(* IEC 61131-3 sources: moqui-plc/iec61131/moqui/framework/src/test/pnp, 17 files *)

(* ---- PickAndPlaceFixture.dut ---- *)
(*#-#-#-#-#-#-#-#-#-#---Declaration---#-#-#-#-#-#-#-#-#-#-#-#-#*)

(* Shared fixture for the pick-and-place test suite *)
TYPE PickAndPlaceFixture : STRUCT
    (* Tripod individual-axis enable flags *)
    tripod1Enable : BOOL;
    tripod2Enable : BOOL;
    tripod3Enable : BOOL;

    (* Tripod coordinated group enable flag *)
    tripodEnable : BOOL;

    (* Drive enable flags *)
    rotaryTableEnable : BOOL;
    conveyorEnable : BOOL;

    (* Tripod TCP position - mirrored from AxisGroup.actualPosition each scan. *)
    tripodActualPos : SM3_Robotics.SMC_POS_REF;

    (* Robot FSM flags *)
    robotState : INT;
    readyForMotion : BOOL; (* Group not in Disabled or ErrorStop *)
    ringAttached : BOOL; (* TRUE while robotState ∈ [70..100] *)
    dontChangePCS_2 : BOOL; (* TRUE while robotState ∈ [90..110] *)
    targetConePtr : POINTER TO Cone; (* Cone targeted during ring-place *)

    (* Environment / conveyor state *)
    activeConePtr : POINTER TO Cone; (* Cone currently defining PCS_2 *)
    ringOnTable : BOOL; (* TRUE if any ring is on the table *)

    (*
     * Coordinate-transform gate.
     * Set TRUE by TripodRobot after MC_SetCoordinateTransform.Done.
     * Prevents re-execution after successful setup.
     *)
    coordTransformDone : BOOL;

    (* Process control flags *)
    automaticPnp : BOOL; (* Continuous automatic pick-and-place cycle *)
    setRing : BOOL; (* Manual one-shot ring release *)

    (* Ring FSM diagnostics - written by Environment each scan *)
    ring1State : DINT;
    ring1TrtDone : BOOL;
    ring1TrtError : BOOL;

    (* Rotary table drive diagnostics - written by Environment each scan *)
    rotaryTableAxisReady : BOOL; (* MC_Power.Status *)
    rotaryTableAxisError : BOOL; (* MC_Power.Error *)
END_STRUCT END_TYPE

(* ---- PickAndPlaceFixture.st ---- *)
(* Shared fixture for the pick-and-place test suite *)
TYPE PickAndPlaceFixture : STRUCT
    (* Tripod individual-axis enable flags *)
    tripod1Enable : BOOL;
    tripod2Enable : BOOL;
    tripod3Enable : BOOL;

    (* Tripod coordinated group enable flag *)
    tripodEnable : BOOL;

    (* Drive enable flags *)
    rotaryTableEnable : BOOL;
    conveyorEnable : BOOL;

    (* Tripod TCP position - mirrored from AxisGroup.actualPosition each scan. *)
    tripodActualPos : SM3_Robotics.SMC_POS_REF;

    (* Robot FSM flags *)
    robotState : INT;
    readyForMotion : BOOL; (* Group not in Disabled or ErrorStop *)
    ringAttached : BOOL; (* TRUE while robotState in [70..100] *)
    dontChangePCS_2 : BOOL; (* TRUE while robotState in [90..110] *)
    targetConePtr : POINTER TO Cone; (* Cone targeted during ring-place *)

    (* Environment / conveyor state *)
    activeConePtr : POINTER TO Cone; (* Cone currently defining PCS_2 *)
    ringOnTable : BOOL; (* TRUE if any ring is on the table *)

    (*
     * Coordinate-transform gate.
     * Set TRUE by TripodRobot after MC_SetCoordinateTransform.Done.
     * Prevents re-execution after successful setup.
     *)
    coordTransformDone : BOOL;

    (* Process control flags *)
    automaticPnp : BOOL; (* Continuous automatic pick-and-place cycle *)
    setRing : BOOL; (* Manual one-shot ring release *)

    (* Ring FSM diagnostics - written by Environment each scan *)
    ring1State : DINT;
    ring1TrtDone : BOOL;
    ring1TrtError : BOOL;

    (* Rotary table drive diagnostics - written by Environment each scan *)
    rotaryTableAxisReady : BOOL; (* MC_Power.Status *)
    rotaryTableAxisError : BOOL; (* MC_Power.Error *)
END_STRUCT END_TYPE

(* ---- PickAndPlaceConsts.gvl ---- *)
(*#-#-#-#-#-#-#-#-#-#---Declaration---#-#-#-#-#-#-#-#-#-#-#-#-#*)

VAR_GLOBAL CONSTANT
    (* Tripod MCS origin - machine-frame → tripod-base transform [mm] *)
    tripodTransX : LREAL := 0;
    tripodTransY : LREAL := 0;
    tripodTransZ : LREAL := 1700;
    tripodSize : LREAL := 180;

    (* Conveyor belt MCS offset *)
    beltTransX : LREAL := 0;
    beltTransY : LREAL := 500;
    beltTransZ : LREAL := 0;

    (* Rotary table MCS offset *)
    tableTransX : LREAL := 0;
    tableTransY : LREAL := -500;
    tableTransZ : LREAL := 0;

    (* TCP offset to bottom of ring (ring thickness + gripper) [mm] *)
    tcpRing : LREAL := 0.02 * tripodSize + 15; (* ≈ 18.6 mm *)

    (* Tripod initial slider positions [mm] *)
    tripod1PosOrig : REAL := 50;
    tripod2PosOrig : REAL := 75;
    tripod3PosOrig : REAL := 25;

    (* Tripod group dynamics *)
    tripodVelocity : LREAL := 1000; (* [mm/s] *)
    tripodAcceleration : LREAL :=  10000; (* [mm/s²] *)
    tripodJerk : LREAL := 100000; (* [mm/s³] *)

    (* Rotary-table drive dynamics *)
    tableVelocity : LREAL :=  50; (* [°/s] *)
    tableAcceleration : LREAL :=  30; (* [°/s²] *)

    (* Conveyor belt drive dynamics *)
    beltVelocity : LREAL := 300; (* [mm/s] *)
    beltAcceleration : LREAL := 150; (* [mm/s²] *)
END_VAR

(* ---- PickAndPlaceConsts.st ---- *)
VAR_GLOBAL CONSTANT
    (* Tripod MCS origin - machine-frame -> tripod-base transform [mm] *)
    tripodTransX : LREAL := 0;
    tripodTransY : LREAL := 0;
    tripodTransZ : LREAL := 1700;
    tripodSize : LREAL := 180;

    (* Conveyor belt MCS offset *)
    beltTransX : LREAL := 0;
    beltTransY : LREAL := 500;
    beltTransZ : LREAL := 0;

    (* Rotary table MCS offset *)
    tableTransX : LREAL := 0;
    tableTransY : LREAL := -500;
    tableTransZ : LREAL := 0;

    (* TCP offset to bottom of ring (ring thickness + gripper) [mm] *)
    tcpRing : LREAL := 0.02 * tripodSize + 15; (* ~= 18.6 mm *)

    (* Tripod initial slider positions [mm] *)
    tripod1PosOrig : REAL := 50;
    tripod2PosOrig : REAL := 75;
    tripod3PosOrig : REAL := 25;

    (* Tripod group dynamics *)
    tripodVelocity : LREAL := 1000; (* [mm/s] *)
    tripodAcceleration : LREAL :=  10000; (* [mm/s²] *)
    tripodJerk : LREAL := 100000; (* [mm/s³] *)

    (* Rotary-table drive dynamics *)
    tableVelocity : LREAL :=  50; (* [°/s] *)
    tableAcceleration : LREAL :=  30; (* [°/s²] *)

    (* Conveyor belt drive dynamics *)
    beltVelocity : LREAL := 300; (* [mm/s] *)
    beltAcceleration : LREAL := 150; (* [mm/s²] *)
END_VAR

(* ---- PickAndPlaceData.gvl ---- *)
(*#-#-#-#-#-#-#-#-#-#---Declaration---#-#-#-#-#-#-#-#-#-#-#-#-#*)

VAR_GLOBAL
    (* Test suite fixture *)
    pnp : PickAndPlaceFixture;
END_VAR

(* ---- PickAndPlaceData.st ---- *)
VAR_GLOBAL
    (* Test suite fixture *)
    pnp : PickAndPlaceFixture;
END_VAR

(* ---- Cone.pou ---- *)
(*#-#-#-#-#-#-#-#-#-#---Declaration---#-#-#-#-#-#-#-#-#-#-#-#-#*)

(* Conveyor-belt cone tracking.
 *
 * FSM:
 *   0   Invisible - waits until previous cone is on belt and far enough,
 *       or 'start' input fires (bootstrap for the first cone)
 *   10  Linking PCS_2 to cone position via MC_TrackConveyorBelt
 *   20  Cone on belt - tracks position until exit point reached
 *)
FUNCTION_BLOCK Cone
VAR_EXTERNAL
	pnp : PickAndPlaceFixture;
END_VAR
VAR_IN_OUT
	activeConePtr : POINTER TO Cone; (* Written to this when cone becomes active *)
END_VAR
VAR_INPUT
	previousConePtr : POINTER TO Cone; (* Previous cone in the circular chain *)
	start : BOOL;
END_VAR
VAR_OUTPUT
	pos : SM3_Robotics.MC_COORD_REF;
	state : DINT;
	onBelt : BOOL;
END_VAR
VAR
	conveyorBeltOrigin : SM3_Robotics.MC_COORD_REF :=
		(X := beltTransX, Y := beltTransY, Z := beltTransZ);
	initialConePosition : SM3_Robotics.MC_COORD_REF := (X := -925, Z := 125);
	tcb : SM3_Robotics.MC_TrackConveyorBelt := (
		ConveyorBeltOrigin := conveyorBeltOrigin,
		InitialObjectPosition := initialConePosition,
		CoordSystem := SM3_Robotics.SMC_COORD_SYSTEM.PCS_2);
	frame : SM3_Robotics.SMC_Frame;
	stateOld : DINT;
END_VAR

(*#-#-#-#-#-#-#-#-#-#---Implementation---#-#-#-#-#-#-#-#-#-#-#-#-#*)

REPEAT
	stateOld := state;

	CASE state OF
		0 :	(* Invisible - wait until the previous cone has advanced sufficiently *)
			IF start OR (NOT pnp.dontChangePCS_2
					AND previousConePtr^.onBelt
					AND previousConePtr^.pos.X >= -250) THEN
				tcb(Execute := FALSE,
					AxisGroup := Tripod,
					ConveyorBelt := DriveConveyorBelt);
				tcb.Execute := TRUE;
				state := state + 10;
			END_IF;

		10 : (* Linking PCS_2 to the position of this cone *)
			IF tcb.Done THEN
				onBelt := TRUE;
				activeConePtr := THIS;
				state := state + 10;
			END_IF;

		20 : (* Cone on belt - track position until it reaches the exit *)
			tcb.cs.GetPose(cs := frame, fTime := Tripod1.fTaskCycle);
			SM3_Robotics.SMC_Frame_To_CoordRef(c := pos, f := frame);
			IF pos.X >= beltTransX + 725 THEN
				onBelt := FALSE;
				state := 0;
			END_IF;
	END_CASE;

	tcb(AxisGroup := Tripod, ConveyorBelt := DriveConveyorBelt);
UNTIL state = stateOld END_REPEAT

(* ---- Cone.st ---- *)
(* Conveyor-belt cone tracking.
 *
 * FSM:
 *   0   Invisible - waits until previous cone is on belt and far enough,
 *       or 'start' input fires (bootstrap for the first cone)
 *   10  Linking PCS_2 to cone position via MC_TrackConveyorBelt
 *   20  Cone on belt - tracks position until exit point reached
 *)
FUNCTION_BLOCK Cone
	VAR_EXTERNAL
		pnp : PickAndPlaceFixture;
	END_VAR
	VAR_IN_OUT
		activeConePtr : POINTER TO Cone; (* Written to this when cone becomes active *)
	END_VAR
	VAR_INPUT
		previousConePtr : POINTER TO Cone; (* Previous cone in the circular chain *)
		start : BOOL;
	END_VAR
	VAR_OUTPUT
		pos : SM3_Robotics.MC_COORD_REF;
		state : DINT;
		onBelt : BOOL;
	END_VAR
	VAR
		conveyorBeltOrigin : SM3_Robotics.MC_COORD_REF :=
			(X := beltTransX, Y := beltTransY, Z := beltTransZ);
		initialConePosition : SM3_Robotics.MC_COORD_REF := (X := -925, Z := 125);
		tcb : SM3_Robotics.MC_TrackConveyorBelt := (
			ConveyorBeltOrigin := conveyorBeltOrigin,
			InitialObjectPosition := initialConePosition,
			CoordSystem := SM3_Robotics.SMC_COORD_SYSTEM.PCS_2);
		frame : SM3_Robotics.SMC_Frame;
		stateOld : DINT;
	END_VAR

	REPEAT
		stateOld := state;

		CASE state OF
			0 :	(* Invisible - wait until the previous cone has advanced sufficiently *)
				IF start OR (NOT pnp.dontChangePCS_2
						AND previousConePtr^.onBelt
						AND previousConePtr^.pos.X >= -250) THEN
					tcb(Execute := FALSE,
						AxisGroup := Tripod,
						ConveyorBelt := DriveConveyorBelt);
					tcb.Execute := TRUE;
					state := state + 10;
				END_IF;

			10 : (* Linking PCS_2 to the position of this cone *)
				IF tcb.Done THEN
					onBelt := TRUE;
					activeConePtr := THIS;
					state := state + 10;
				END_IF;

			20 : (* Cone on belt - track position until it reaches the exit *)
				tcb.cs.GetPose(cs := frame, fTime := Tripod1.fTaskCycle);
				SM3_Robotics.SMC_Frame_To_CoordRef(c := pos, f := frame);
				IF pos.X >= beltTransX + 725 THEN
					onBelt := FALSE;
					state := 0;
				END_IF;
		END_CASE;

		tcb(AxisGroup := Tripod, ConveyorBelt := DriveConveyorBelt);
	UNTIL state = stateOld END_REPEAT
	END_FUNCTION_BLOCK

(* ---- Environment.pou ---- *)
(*#-#-#-#-#-#-#-#-#-#---Declaration---#-#-#-#-#-#-#-#-#-#-#-#-#*)

{attribute 'no_assign'}
(* Hardware-abstraction layer for the conveyance environment.
 *
 * Responsibilities:
 *   1. Drive the rotary-table and conveyor-belt axes with MC_Power + MC_MoveVelocity.
 *      (continuous rotation/feed - no homing required for these drives).
 *   2. Run the cone state machines (three cones on the conveyor belt).
 *   3. Run the ring state machines (two rings on the rotary table).
 *   4. Publish activeCone and ringOnTable each scan.
 *)
FUNCTION_BLOCK Environment
VAR_EXTERNAL
	pnp : PickAndPlaceFixture;
END_VAR
VAR_INPUT
	operationType : OperatingMode;
END_VAR
VAR
	(* Drive axes - MC_Power + MC_MoveVelocity, no homing for continuous drives *)
	powRotaryTable : MC_Power := (Enable := TRUE, bRegulatorOn := TRUE, bDriveStart := TRUE);
	powConveyorBelt : MC_Power := (Enable := TRUE, bRegulatorOn := TRUE, bDriveStart := TRUE);
	mvRotaryTable : MC_MoveVelocity := (Execute := TRUE, Velocity := tableVelocity, Acceleration := tableAcceleration, Deceleration := tableAcceleration, Jerk := 1000);
	mvConveyorBelt : MC_MoveVelocity := (Execute := TRUE, Velocity := beltVelocity, Acceleration := beltAcceleration, Deceleration := beltAcceleration, Jerk := 1000);

	(* Cones - three instances on the belt (circular chain) *)
	cone1 : Cone;
	cone2 : Cone;
	cone3 : Cone;

	(* Rings - two instances on the rotary table *)
	ring1 : Ring;
	ring2 : Ring;

	ring1StartPos : SM3_Robotics.MC_COORD_REF := (X :=  75, Y := 100, Z := 0);
	ring2StartPos : SM3_Robotics.MC_COORD_REF := (X := -75, Y := 100, Z := 0);

	init : BOOL := TRUE; (* First-scan bootstrap flag *)
END_VAR

(*#-#-#-#-#-#-#-#-#-#---Implementation---#-#-#-#-#-#-#-#-#-#-#-#-#*)

(* Rotary table and conveyor belt drives - power and continuous velocity *)
powRotaryTable(Axis := DriveRotaryTable);
powConveyorBelt(Axis := DriveConveyorBelt);

(* Drive status diagnostics - updated before the guard so they are visible even if RETURN fires *)
pnp.rotaryTableAxisReady := powRotaryTable.Status;
pnp.rotaryTableAxisError := powRotaryTable.Error;

(* Wait for both drives powered before running cones / rings *)
IF NOT (powRotaryTable.Status AND powConveyorBelt.Status) THEN
	init := TRUE;
	RETURN;
END_IF;
mvRotaryTable(Axis := DriveRotaryTable);
mvConveyorBelt(Axis := DriveConveyorBelt);

(* Wait for the tripod group to be ready before starting cone/ring FSMs *)
IF NOT pnp.readyForMotion THEN
	RETURN;
END_IF;

(* Cone state machines *)
(*
 * cone1.start := init bootstraps the circular chain on the first scan:
 *   cone1 activates immediately (skips the chain-guard condition).
 *   cone2 and cone3 activate in sequence once cone1 advances on the belt.
 *)
cone1(activeConePtr := pnp.activeConePtr, previousConePtr := ADR(cone3), start := init);
cone2(activeConePtr := pnp.activeConePtr, previousConePtr := ADR(cone1), start := FALSE);
cone3(activeConePtr := pnp.activeConePtr, previousConePtr := ADR(cone2), start := FALSE);

(* Ring state machines *)
IF init THEN
	ring1.startPos := ring1StartPos;
	ring2.startPos := ring2StartPos;
END_IF;

ring1(otherRingPtr := ADR(ring2));
ring2(otherRingPtr := ADR(ring1));

(* Publish environment state to pnp *)
pnp.ringOnTable := ring1.onTable OR ring2.onTable;

(* Ring FSM diagnostics *)
pnp.ring1State := ring1.state;
pnp.ring1TrtDone := ring1.trt.Done;
pnp.ring1TrtError := ring1.trt.Error;

init := FALSE;

(* ---- Environment.st ---- *)
(* Hardware-abstraction layer for the conveyance environment.
 *
 * Responsibilities:
 *   1. Drive the rotary-table and conveyor-belt axes with MC_Power + MC_MoveVelocity.
 *      (continuous rotation/feed - no homing required for these drives).
 *   2. Run the cone state machines (three cones on the conveyor belt).
 *   3. Run the ring state machines (two rings on the rotary table).
 *   4. Publish activeCone and ringOnTable each scan.
 *)
FUNCTION_BLOCK Environment
	VAR_EXTERNAL
		pnp : PickAndPlaceFixture;
	END_VAR
	VAR_INPUT
		operationType : OperatingMode;
	END_VAR
	VAR
		(* Drive axes - MC_Power + MC_MoveVelocity, no homing for continuous drives *)
		powRotaryTable : MC_Power := (Enable := TRUE, bRegulatorOn := TRUE, bDriveStart := TRUE);
		powConveyorBelt : MC_Power := (Enable := TRUE, bRegulatorOn := TRUE, bDriveStart := TRUE);
		mvRotaryTable : MC_MoveVelocity := (Execute := TRUE, Velocity := tableVelocity, Acceleration := tableAcceleration, Deceleration := tableAcceleration, Jerk := 1000);
		mvConveyorBelt : MC_MoveVelocity := (Execute := TRUE, Velocity := beltVelocity, Acceleration := beltAcceleration, Deceleration := beltAcceleration, Jerk := 1000);

		(* Cones - three instances on the belt (circular chain) *)
		cone1 : Cone;
		cone2 : Cone;
		cone3 : Cone;

		(* Rings - two instances on the rotary table *)
		ring1 : Ring;
		ring2 : Ring;

		ring1StartPos : SM3_Robotics.MC_COORD_REF := (X :=  75, Y := 100, Z := 0);
		ring2StartPos : SM3_Robotics.MC_COORD_REF := (X := -75, Y := 100, Z := 0);

		init : BOOL := TRUE; (* First-scan bootstrap flag *)
	END_VAR

	(* Rotary table and conveyor belt drives - power and continuous velocity *)
	powRotaryTable(Axis := DriveRotaryTable);
	powConveyorBelt(Axis := DriveConveyorBelt);

	(* Drive status diagnostics - updated before the guard so they are visible even if RETURN fires *)
	pnp.rotaryTableAxisReady := powRotaryTable.Status;
	pnp.rotaryTableAxisError := powRotaryTable.Error;

	(* Wait for both drives powered before running cones / rings *)
	IF NOT (powRotaryTable.Status AND powConveyorBelt.Status) THEN
		init := TRUE;
		RETURN;
	END_IF;
	mvRotaryTable(Axis := DriveRotaryTable);
	mvConveyorBelt(Axis := DriveConveyorBelt);

	(* Wait for the tripod group to be ready before starting cone/ring FSMs *)
	IF NOT pnp.readyForMotion THEN
		RETURN;
	END_IF;

	(* Cone state machines *)
	(*
	 * cone1.start := init bootstraps the circular chain on the first scan:
	 *   cone1 activates immediately (skips the chain-guard condition).
	 *   cone2 and cone3 activate in sequence once cone1 advances on the belt.
	 *)
	cone1(activeConePtr := pnp.activeConePtr, previousConePtr := ADR(cone3), start := init);
	cone2(activeConePtr := pnp.activeConePtr, previousConePtr := ADR(cone1), start := FALSE);
	cone3(activeConePtr := pnp.activeConePtr, previousConePtr := ADR(cone2), start := FALSE);

	(* Ring state machines *)
	IF init THEN
		ring1.startPos := ring1StartPos;
		ring2.startPos := ring2StartPos;
	END_IF;

	ring1(otherRingPtr := ADR(ring2));
	ring2(otherRingPtr := ADR(ring1));

	(* Publish environment state to pnp *)
	pnp.ringOnTable := ring1.onTable OR ring2.onTable;

	(* Ring FSM diagnostics *)
	pnp.ring1State := ring1.state;
	pnp.ring1TrtDone := ring1.trt.Done;
	pnp.ring1TrtError := ring1.trt.Error;

	init := FALSE;
	END_FUNCTION_BLOCK

(* ---- Ring.pou ---- *)
(*#-#-#-#-#-#-#-#-#-#---Declaration---#-#-#-#-#-#-#-#-#-#-#-#-#*)

(* Rotary-table ring tracking.
 *
 * State machine:
 *   0   Ring at start position - waits for safe conditions + trigger
 *   10  Linking PCS_1 to ring via MC_TrackRotaryTable
 *   20  Ring on table, spinning - waits until robot is free
 *   30  Waiting for robot to pick up ring
 *   40  Ring attached to robot - follows TCP position
 *   50  Ring placed on cone - follows cone position until cone leaves belt
 *)
FUNCTION_BLOCK Ring
VAR_EXTERNAL
	pnp : PickAndPlaceFixture;
END_VAR
VAR_INPUT
	otherRingPtr : POINTER TO Ring; (* The other ring in the pair *)
	startPos : SM3_Robotics.MC_COORD_REF; (* Initial position in MCS *)
END_VAR
VAR_OUTPUT
	pos : SM3_Robotics.MC_COORD_REF;
	state  : DINT;
	onTable : BOOL;
END_VAR
VAR
	stateOld : DINT;
	frame : SM3_Robotics.SMC_Frame;
	rotaryTableOrigin : SM3_Robotics.MC_COORD_REF :=
		(X := tableTransX, Y := tableTransY, Z := tableTransZ);
	initialObjectPosition : SM3_Robotics.MC_COORD_REF := (Y := 400, Z := 30);
	trt : SM3_Robotics.MC_TrackRotaryTable := (
		RotaryTableOrigin := rotaryTableOrigin,
		initialObjectPosition := initialObjectPosition,
		CoordSystem := SM3_Robotics.SMC_COORD_SYSTEM.PCS_1);
	conePtr : POINTER TO Cone;
END_VAR

(*#-#-#-#-#-#-#-#-#-#---Implementation---#-#-#-#-#-#-#-#-#-#-#-#-#*)

REPEAT
	stateOld := state;
	CASE state OF

	0 :	(* Ring at start position - wait for safe conditions and cycle trigger *)
		pos := startPos;

		IF pnp.readyForMotion AND (otherRingPtr^.state = 0 OR otherRingPtr^.state >= 40)
				AND (pnp.setRing OR pnp.automaticPnp) THEN
			trt(Execute := FALSE,
			    AxisGroup := Tripod,
			    RotaryTable := DriveRotaryTable);
			trt.Execute := TRUE;
			state := state + 10;
		END_IF;

	10 : (* Linking PCS_1 to the position of this ring *)
		IF trt.Done THEN
			state := state + 10;
		END_IF;

	20 : (* Ring on rotary table, spinning - wait until robot is free to pick *)
		trt.cs.GetPose(cs := frame, fTime := Tripod1.fTaskCycle);
		SM3_Robotics.SMC_Frame_To_CoordRef(c := pos, f := frame);

		IF NOT pnp.ringAttached THEN
			state := state + 10;
		END_IF;

	30 : (* Waiting for robot to attach to ring *)
		trt.cs.GetPose(cs := frame, fTime := Tripod1.fTaskCycle);
		SM3_Robotics.SMC_Frame_To_CoordRef(c := pos, f := frame);

		IF pnp.ringAttached THEN
			state := state + 10;
		END_IF;

	40 : (* Ring attached to robot - follow TCP position *)
		pos.X := pnp.tripodActualPos.c.X;
		pos.Y := pnp.tripodActualPos.c.Y;
		pos.Z := pnp.tripodActualPos.c.Z - tcpRing;

		IF NOT pnp.ringAttached THEN
			conePtr := pnp.targetConePtr;
			state := state + 10;
		END_IF;

	50 : (* Ring placed on cone - follow cone position until cone exits belt *)
		pos.X := conePtr^.pos.X;
		pos.Y := conePtr^.pos.Y;
		pos.Z := conePtr^.pos.Z;

		IF NOT conePtr^.onBelt THEN
			state := 0;
		END_IF;
	END_CASE;

	trt(AxisGroup := Tripod, RotaryTable := DriveRotaryTable);
UNTIL state = stateOld END_REPEAT;

onTable := state = 20 OR state = 30;

(* ---- Ring.st ---- *)
(* Rotary-table ring tracking.
 *
 * State machine:
 *   0   Ring at start position - waits for safe conditions + trigger
 *   10  Linking PCS_1 to ring via MC_TrackRotaryTable
 *   20  Ring on table, spinning - waits until robot is free
 *   30  Waiting for robot to pick up ring
 *   40  Ring attached to robot - follows TCP position
 *   50  Ring placed on cone - follows cone position until cone leaves belt
 *)
FUNCTION_BLOCK Ring
	VAR_EXTERNAL
		pnp : PickAndPlaceFixture;
	END_VAR
	VAR_INPUT
		otherRingPtr : POINTER TO Ring; (* The other ring in the pair *)
		startPos : SM3_Robotics.MC_COORD_REF; (* Initial position in MCS *)
	END_VAR
	VAR_OUTPUT
		pos : SM3_Robotics.MC_COORD_REF;
		state  : DINT;
		onTable : BOOL;
	END_VAR
	VAR
		stateOld : DINT;
		frame : SM3_Robotics.SMC_Frame;
		rotaryTableOrigin : SM3_Robotics.MC_COORD_REF :=
			(X := tableTransX, Y := tableTransY, Z := tableTransZ);
		initialObjectPosition : SM3_Robotics.MC_COORD_REF := (Y := 400, Z := 30);
		trt : SM3_Robotics.MC_TrackRotaryTable := (
			RotaryTableOrigin := rotaryTableOrigin,
			initialObjectPosition := initialObjectPosition,
			CoordSystem := SM3_Robotics.SMC_COORD_SYSTEM.PCS_1);
		conePtr : POINTER TO Cone;
	END_VAR

	REPEAT
		stateOld := state;
		CASE state OF

		0 :	(* Ring at start position - wait for safe conditions and cycle trigger *)
			pos := startPos;

			IF pnp.readyForMotion AND (otherRingPtr^.state = 0 OR otherRingPtr^.state >= 40)
					AND (pnp.setRing OR pnp.automaticPnp) THEN
				trt(Execute := FALSE,
				    AxisGroup := Tripod,
				    RotaryTable := DriveRotaryTable);
				trt.Execute := TRUE;
				state := state + 10;
			END_IF;

		10 : (* Linking PCS_1 to the position of this ring *)
			IF trt.Done THEN
				state := state + 10;
			END_IF;

		20 : (* Ring on rotary table, spinning - wait until robot is free to pick *)
			trt.cs.GetPose(cs := frame, fTime := Tripod1.fTaskCycle);
			SM3_Robotics.SMC_Frame_To_CoordRef(c := pos, f := frame);

			IF NOT pnp.ringAttached THEN
				state := state + 10;
			END_IF;

		30 : (* Waiting for robot to attach to ring *)
			trt.cs.GetPose(cs := frame, fTime := Tripod1.fTaskCycle);
			SM3_Robotics.SMC_Frame_To_CoordRef(c := pos, f := frame);

			IF pnp.ringAttached THEN
				state := state + 10;
			END_IF;

		40 : (* Ring attached to robot - follow TCP position *)
			pos.X := pnp.tripodActualPos.c.X;
			pos.Y := pnp.tripodActualPos.c.Y;
			pos.Z := pnp.tripodActualPos.c.Z - tcpRing;

			IF NOT pnp.ringAttached THEN
				conePtr := pnp.targetConePtr;
				state := state + 10;
			END_IF;

		50 : (* Ring placed on cone - follow cone position until cone exits belt *)
			pos.X := conePtr^.pos.X;
			pos.Y := conePtr^.pos.Y;
			pos.Z := conePtr^.pos.Z;

			IF NOT conePtr^.onBelt THEN
				state := 0;
			END_IF;
		END_CASE;

		trt(AxisGroup := Tripod, RotaryTable := DriveRotaryTable);
	UNTIL state = stateOld END_REPEAT;

	onTable := state = 20 OR state = 30;
	END_FUNCTION_BLOCK

(* ---- TripodRobot.pou ---- *)
(*#-#-#-#-#-#-#-#-#-#---Declaration---#-#-#-#-#-#-#-#-#-#-#-#-#*)

{attribute 'no_assign'}
(* Tripod robot motion FSM using Moqui AxisGroup and Axis wrappers.
 *
 * FSM:
 *   0    Wait for all three tripod axes powered and ready
 *   10   Set initial slider positions (AxisCmd.SetPosition x 3)
 *   20   Set MCS coordinate transform (MC_SetCoordinateTransform, direct)
 *   30   Enable axis group (AxisGroup.groupEnable -> Standby)
 *   40   Wait for ring on table; issue MoveLinearAbsolute to ring (PCS_1)
 *   50   Wait commandExecuted (arrival at ring)
 *   60   Wait 200 ms (ring following), then issue MoveLinearRelative upward (PCS_1)
 *   70   Wait commandExecuted; issue MoveLinearAbsolute to rest (WCS)
 *   80   Wait commandExecuted; [release] then MoveLinearAbsolute above cone (PCS_2)
 *   90   Wait commandExecuted; [release] then MoveLinearAbsolute on cone (PCS_2)
 *   100  Wait commandExecuted; [release] then MoveLinearAbsolute above cone (PCS_2)
 *   110  Wait commandExecuted; [release] then MoveLinearAbsolute to rest (WCS)
 *   120  Wait commandExecuted; [release] then loop to state 40
 *
 * [release] means: the previous command was also MoveLinearAbsolute, so the
 * AxisGroup FSM stays in CheckLinearAbsoluteState (commandExecuted=TRUE) until the caller changes cmd.
 * On commandExecuted, set cmd=Idle -> AxisGroup returns to Standby (ready=TRUE) -> set the new MoveLinearAbsolute target.
 * This 2-scan handshake is needed only when two consecutive commands share the
 * same AxisGroupCmd value (both MoveLinearAbsolute).
 *
 * Unconditional FB calls at the bottom execute every scan regardless of state,
 * following the standard CODESYS PLCopen pattern.
 *)
FUNCTION_BLOCK TripodRobot
VAR_EXTERNAL
	pnp : PickAndPlaceFixture;
END_VAR
VAR_INPUT
	operationType : OperatingMode;
END_VAR
VAR_OUTPUT
	groupError : BOOL;
	groupErrorId : DWORD;
END_VAR
VAR
	(* Tripod individual axes *)
	tripodAxis1 : Axis;
	tripodAxis2 : Axis;
	tripodAxis3 : Axis;

	(* Tripod coordinated group - AxisGroup wraps all Cartesian moves *)
	tripodGroup : AxisGroup;

	(* Coordinate transform - direct PLCopen call *)
	setCoord : SM3_Robotics.MC_SetCoordinateTransform;
	mcs : SM3_Robotics.MC_COORD_REF;

	(* 200ms ring-following timer (state 60) *)
	ton : TON := (PT := T#200MS);

	(*
     * Constant Cartesian target positions.
	 * All X,Y components default to 0 (struct zero-init).
	 * Only Z (and coordinate system) distinguishes them.
     *)
	posAboveRingPCS1 : SM3_Robotics.SMC_POS_REF; (* Z = tcpRing, PCS_1 *)
	posAboveConePCS2 : SM3_Robotics.SMC_POS_REF; (* Z = 200, PCS_2 *)
	posOnConePCS2 : SM3_Robotics.SMC_POS_REF; (* Z = tcpRing, PCS_2 *)
	posRestWCS : SM3_Robotics.SMC_POS_REF; (* Z = 300, WCS *)
END_VAR

(*#-#-#-#-#-#-#-#-#-#---Implementation---#-#-#-#-#-#-#-#-#-#-#-#-#*)

(* Target positions - set each scan (struct re-init on first scan) *)
posAboveRingPCS1.c.Z := tcpRing;
posAboveConePCS2.c.Z := 200;
posOnConePCS2.c.Z := tcpRing;
posRestWCS.c.Z := 300;

(* Tripod robot FSM *)
CASE pnp.robotState OF
	0 : (* Wait for all three tripod axes powered and homed *)
		pnp.tripod1Enable := TRUE;
		pnp.tripod2Enable := TRUE;
		pnp.tripod3Enable := TRUE;
		IF tripodAxis1.ready AND tripodAxis2.ready AND tripodAxis3.ready THEN
			pnp.robotState := 10;
		END_IF

	10 : (* Set initial slider positions *)
		tripodAxis1.cmd := AxisCmd.SetPosition;
		tripodAxis1.position := tripod1PosOrig;
		tripodAxis2.cmd := AxisCmd.SetPosition;
		tripodAxis2.position := tripod2PosOrig;
		tripodAxis3.cmd := AxisCmd.SetPosition;
		tripodAxis3.position := tripod3PosOrig;

		IF tripodAxis1.commandExecuted AND tripodAxis2.commandExecuted
				AND tripodAxis3.commandExecuted THEN
			tripodAxis1.cmd := AxisCmd.Idle;
			tripodAxis2.cmd := AxisCmd.Idle;
			tripodAxis3.cmd := AxisCmd.Idle;
			setCoord.Execute := FALSE; (* Arm rising edge for state 20 *)
			pnp.robotState := 20;
		END_IF;

	20 : (* Set MCS coordinate transform (direct MC_SetCoordinateTransform) *)
		mcs.X := tripodTransX;
		mcs.Y := tripodTransY;
		mcs.Z := tripodTransZ;
		setCoord.Execute := TRUE;
		setCoord.CoordTransform := mcs;
		setCoord.CoordSystem := SM3_Robotics.SMC_COORD_SYSTEM.MCS;

		IF setCoord.Done THEN
			pnp.coordTransformDone := TRUE;
			pnp.robotState := 30;
		END_IF;

	30 : (* Enable axis group - AxisGroup transitions to Standby *)
		pnp.tripodEnable := TRUE;

		IF tripodGroup.ready THEN
			pnp.robotState := 40;
		END_IF;

	40 : (* Wait for ring on table, then issue move to ring (PCS_1) *)
		IF pnp.ringOnTable THEN
			tripodGroup.cmd := AxisGroupCmd.MoveLinearAbsolute;
			tripodGroup.endPoint := posAboveRingPCS1;
			tripodGroup.coordinateSystem := SM3_Robotics.SMC_COORD_SYSTEM.PCS_1;
			tripodGroup.velocity := tripodVelocity;
			tripodGroup.acceleration := tripodAcceleration;
			tripodGroup.deceleration := tripodAcceleration;
			tripodGroup.jerk := tripodJerk;
			tripodGroup.bufferMode := SM3_Basic.MC_BUFFER_MODE.BlendingHigh;
			tripodGroup.transitionMode := SM3_Robotics.MC_TRANSITION_MODE.TMCornerDistance;
			tripodGroup.transitionParameter := 500;
			pnp.robotState := 50;
		END_IF;

	50 : (* Wait for arrival at ring *)
		IF tripodGroup.commandExecuted THEN
			ton(IN := FALSE); (* Reset 200 ms timer *)
			pnp.robotState := 60;
		END_IF;

	60 : (* Wait 200 ms following the ring, then move upward *)
		ton(IN := TRUE);

		IF ton.Q THEN
			tripodGroup.cmd := AxisGroupCmd.MoveLinearRelative;
			tripodGroup.endPoint.c.X := 0;
			tripodGroup.endPoint.c.Y := 0;
			tripodGroup.endPoint.c.Z := 150;
			tripodGroup.coordinateSystem := SM3_Robotics.SMC_COORD_SYSTEM.WCS;
			tripodGroup.bufferMode := SM3_Basic.MC_BUFFER_MODE.Buffered;
			tripodGroup.transitionMode := SM3_Robotics.MC_TRANSITION_MODE.TMNone;
			tripodGroup.transitionParameter := 0;
			pnp.robotState := 70;
		END_IF;

	70 : (* Queue MoveLinearAbsolute to rest (WCS), matching the sample's buffered handoff *)
		tripodGroup.cmd := AxisGroupCmd.MoveLinearAbsolute;
		tripodGroup.endPoint := posRestWCS;
		tripodGroup.coordinateSystem := SM3_Robotics.SMC_COORD_SYSTEM.WCS;
		tripodGroup.bufferMode := SM3_Basic.MC_BUFFER_MODE.BlendingHigh;
		tripodGroup.transitionMode := SM3_Robotics.MC_TRANSITION_MODE.TMCornerDistance;
		tripodGroup.transitionParameter := 500;
		pnp.robotState := 80;

	80 : (* [release] wait rest-pos done; then move above cone (PCS_2) *)
		IF tripodGroup.commandExecuted THEN
			tripodGroup.cmd := AxisGroupCmd.Idle;
		ELSIF tripodGroup.ready THEN
			pnp.targetConePtr := pnp.activeConePtr;
			tripodGroup.cmd := AxisGroupCmd.MoveLinearAbsolute;
			tripodGroup.endPoint := posAboveConePCS2;
			tripodGroup.coordinateSystem := SM3_Robotics.SMC_COORD_SYSTEM.PCS_2;
			tripodGroup.bufferMode := SM3_Basic.MC_BUFFER_MODE.aborting;
			tripodGroup.transitionMode := SM3_Robotics.MC_TRANSITION_MODE.TMNone;
			tripodGroup.transitionParameter := 0;
			pnp.robotState := 90;
		END_IF;

	90 : (* [release] wait above-cone done; then move down to cone (PCS_2) *)
		IF tripodGroup.commandExecuted THEN
			tripodGroup.cmd := AxisGroupCmd.Idle;
		ELSIF tripodGroup.ready THEN
			tripodGroup.cmd := AxisGroupCmd.MoveLinearAbsolute;
			tripodGroup.endPoint := posOnConePCS2;
			tripodGroup.coordinateSystem := SM3_Robotics.SMC_COORD_SYSTEM.PCS_2;
			tripodGroup.bufferMode := SM3_Basic.MC_BUFFER_MODE.aborting;
			tripodGroup.transitionMode := SM3_Robotics.MC_TRANSITION_MODE.TMNone;
			tripodGroup.transitionParameter := 0;
			pnp.robotState := 100;
		END_IF;

	100 : (* [release] ring placed on cone; move back above cone (PCS_2) *)
		IF tripodGroup.commandExecuted THEN
			tripodGroup.cmd := AxisGroupCmd.Idle;
		ELSIF tripodGroup.ready THEN
			tripodGroup.cmd := AxisGroupCmd.MoveLinearAbsolute;
			tripodGroup.endPoint := posAboveConePCS2;
			tripodGroup.coordinateSystem := SM3_Robotics.SMC_COORD_SYSTEM.PCS_2;
			tripodGroup.bufferMode := SM3_Basic.MC_BUFFER_MODE.Buffered;
			tripodGroup.transitionMode := SM3_Robotics.MC_TRANSITION_MODE.TMNone;
			tripodGroup.transitionParameter := 0;
			pnp.robotState := 110;
		END_IF;

	110 : (* [release] wait above-cone done; move back to rest (WCS) *)
		IF tripodGroup.commandExecuted THEN
			tripodGroup.cmd := AxisGroupCmd.Idle;
		ELSIF tripodGroup.ready THEN
			tripodGroup.cmd := AxisGroupCmd.MoveLinearAbsolute;
			tripodGroup.endPoint := posRestWCS;
			tripodGroup.coordinateSystem := SM3_Robotics.SMC_COORD_SYSTEM.WCS;
			tripodGroup.bufferMode := SM3_Basic.MC_BUFFER_MODE.aborting;
			tripodGroup.transitionMode := SM3_Robotics.MC_TRANSITION_MODE.TMNone;
			tripodGroup.transitionParameter := 0;
			pnp.robotState := 120;
		END_IF;

	120 : (* [release] cycle complete; loop to state 40 *)
		IF tripodGroup.commandExecuted THEN
			tripodGroup.cmd := AxisGroupCmd.Idle;
		ELSIF tripodGroup.ready THEN
			pnp.robotState := 40;
		END_IF;
END_CASE;

(* Mirror TCP position to shared parameters *)
pnp.tripodActualPos := tripodGroup.actualPosition;

(* Status flags (read by Ring and Cone) *)
pnp.readyForMotion := NOT tripodGroup.groupError AND tripodGroup.status <> AxisGroupStatus.Disabled;
pnp.ringAttached := pnp.robotState >= 70 AND pnp.robotState <= 100;
pnp.dontChangePCS_2 := pnp.robotState >= 90 AND pnp.robotState <= 110;

groupError := tripodGroup.groupError;
groupErrorId := tripodGroup.groupErrorId;

(* Auto-reset: rising edge on first scan groupError is TRUE triggers MC_GroupReset → Standby *)
tripodGroup.reset := tripodGroup.groupError;

(* Individual tripod axes *)
tripodAxis1(
	slave := Tripod1,
	axisEnable := pnp.tripod1Enable,
	cmd := tripodAxis1.cmd,
	position := tripodAxis1.position,
	velocity := tripodVelocity,
	acceleration := tripodAcceleration,
	deceleration := tripodAcceleration,
	jerk := tripodJerk);

tripodAxis2(
	slave := Tripod2,
	axisEnable := pnp.tripod2Enable,
	cmd := tripodAxis2.cmd,
	position := tripodAxis2.position,
	velocity := tripodVelocity,
	acceleration := tripodAcceleration,
	deceleration := tripodAcceleration,
	jerk := tripodJerk);

tripodAxis3(
	slave := Tripod3,
	axisEnable := pnp.tripod3Enable,
	cmd := tripodAxis3.cmd,
	position := tripodAxis3.position,
	velocity := tripodVelocity,
	acceleration := tripodAcceleration,
	deceleration := tripodAcceleration,
	jerk := tripodJerk);

(* Coordinated tripod group - AxisGroup.pou *)
tripodGroup(
	axisGroupId := 'Tripod',
	axisGroupName := 'Tripod',
	group := Tripod,
	groupEnable := pnp.tripodEnable);

(* Coordinate transform - called every scan so the FB processes its internal state machine *)
setCoord(AxisGroup := Tripod);

(* ---- TripodRobot.st ---- *)
(* Tripod robot motion FSM using Moqui AxisGroup and Axis wrappers.
 *
 * FSM:
 *   0    Wait for all three tripod axes powered and ready
 *   10   Set initial slider positions (AxisCmd.SetPosition x 3)
 *   20   Set MCS coordinate transform (MC_SetCoordinateTransform, direct)
 *   30   Enable axis group (AxisGroup.groupEnable -> Standby)
 *   40   Wait for ring on table; issue MoveLinearAbsolute to ring (PCS_1)
 *   50   Wait commandExecuted (arrival at ring)
 *   60   Wait 200 ms (ring following), then issue MoveLinearRelative upward (PCS_1)
 *   70   Wait commandExecuted; issue MoveLinearAbsolute to rest (WCS)
 *   80   Wait commandExecuted; [release] then MoveLinearAbsolute above cone (PCS_2)
 *   90   Wait commandExecuted; [release] then MoveLinearAbsolute on cone (PCS_2)
 *   100  Wait commandExecuted; [release] then MoveLinearAbsolute above cone (PCS_2)
 *   110  Wait commandExecuted; [release] then MoveLinearAbsolute to rest (WCS)
 *   120  Wait commandExecuted; [release] then loop to state 40
 *
 * [release] means: the previous command was also MoveLinearAbsolute, so the
 * AxisGroup FSM stays in CheckLinearAbsoluteState (commandExecuted=TRUE) until the caller changes cmd.
 * On commandExecuted, set cmd=Idle -> AxisGroup returns to Standby (ready=TRUE) -> set the new MoveLinearAbsolute target.
 * This 2-scan handshake is needed only when two consecutive commands share the
 * same AxisGroupCmd value (both MoveLinearAbsolute).
 *
 * Unconditional FB calls at the bottom execute every scan regardless of state,
 * following the standard CODESYS PLCopen pattern.
 *)
FUNCTION_BLOCK TripodRobot
	VAR_EXTERNAL
		pnp : PickAndPlaceFixture;
	END_VAR
	VAR_INPUT
		operationType : OperatingMode;
	END_VAR
	VAR_OUTPUT
		groupError : BOOL;
		groupErrorId : DWORD;
	END_VAR
	VAR
		(* Tripod individual axes *)
		tripodAxis1 : Axis;
		tripodAxis2 : Axis;
		tripodAxis3 : Axis;

		(* Tripod coordinated group - AxisGroup wraps all Cartesian moves *)
		tripodGroup : AxisGroup;

		(* Coordinate transform - direct PLCopen call *)
		setCoord : SM3_Robotics.MC_SetCoordinateTransform;
		mcs : SM3_Robotics.MC_COORD_REF;

		(* 200ms ring-following timer (state 60) *)
		ton : TON := (PT := T#200MS);

		(*
	     * Constant Cartesian target positions.
		 * All X,Y components default to 0 (struct zero-init).
		 * Only Z (and coordinate system) distinguishes them.
	     *)
		posAboveRingPCS1 : SM3_Robotics.SMC_POS_REF; (* Z = tcpRing, PCS_1 *)
		posAboveConePCS2 : SM3_Robotics.SMC_POS_REF; (* Z = 200, PCS_2 *)
		posOnConePCS2 : SM3_Robotics.SMC_POS_REF; (* Z = tcpRing, PCS_2 *)
		posRestWCS : SM3_Robotics.SMC_POS_REF; (* Z = 300, WCS *)
	END_VAR

	(* Target positions - set each scan (struct re-init on first scan) *)
	posAboveRingPCS1.c.Z := tcpRing;
	posAboveConePCS2.c.Z := 200;
	posOnConePCS2.c.Z := tcpRing;
	posRestWCS.c.Z := 300;

	(* Tripod robot FSM *)
	CASE pnp.robotState OF
		0 : (* Wait for all three tripod axes powered and homed *)
			pnp.tripod1Enable := TRUE;
			pnp.tripod2Enable := TRUE;
			pnp.tripod3Enable := TRUE;
			IF tripodAxis1.ready AND tripodAxis2.ready AND tripodAxis3.ready THEN
				pnp.robotState := 10;
			END_IF

		10 : (* Set initial slider positions *)
			tripodAxis1.cmd := AxisCmd.SetPosition;
			tripodAxis1.position := tripod1PosOrig;
			tripodAxis2.cmd := AxisCmd.SetPosition;
			tripodAxis2.position := tripod2PosOrig;
			tripodAxis3.cmd := AxisCmd.SetPosition;
			tripodAxis3.position := tripod3PosOrig;

			IF tripodAxis1.commandExecuted AND tripodAxis2.commandExecuted
					AND tripodAxis3.commandExecuted THEN
				tripodAxis1.cmd := AxisCmd.Idle;
				tripodAxis2.cmd := AxisCmd.Idle;
				tripodAxis3.cmd := AxisCmd.Idle;
				setCoord.Execute := FALSE; (* Arm rising edge for state 20 *)
				pnp.robotState := 20;
			END_IF;

		20 : (* Set MCS coordinate transform (direct MC_SetCoordinateTransform) *)
			mcs.X := tripodTransX;
			mcs.Y := tripodTransY;
			mcs.Z := tripodTransZ;
			setCoord.Execute := TRUE;
			setCoord.CoordTransform := mcs;
			setCoord.CoordSystem := SM3_Robotics.SMC_COORD_SYSTEM.MCS;

			IF setCoord.Done THEN
				pnp.coordTransformDone := TRUE;
				pnp.robotState := 30;
			END_IF;

		30 : (* Enable axis group - AxisGroup transitions to Standby *)
			pnp.tripodEnable := TRUE;

			IF tripodGroup.ready THEN
				pnp.robotState := 40;
			END_IF;

		40 : (* Wait for ring on table, then issue move to ring (PCS_1) *)
			IF pnp.ringOnTable THEN
				tripodGroup.cmd := AxisGroupCmd.MoveLinearAbsolute;
				tripodGroup.endPoint := posAboveRingPCS1;
				tripodGroup.coordinateSystem := SM3_Robotics.SMC_COORD_SYSTEM.PCS_1;
				tripodGroup.velocity := tripodVelocity;
				tripodGroup.acceleration := tripodAcceleration;
				tripodGroup.deceleration := tripodAcceleration;
				tripodGroup.jerk := tripodJerk;
				tripodGroup.bufferMode := SM3_Basic.MC_BUFFER_MODE.BlendingHigh;
				tripodGroup.transitionMode := SM3_Robotics.MC_TRANSITION_MODE.TMCornerDistance;
				tripodGroup.transitionParameter := 500;
				pnp.robotState := 50;
			END_IF;

		50 : (* Wait for arrival at ring *)
			IF tripodGroup.commandExecuted THEN
				ton(IN := FALSE); (* Reset 200 ms timer *)
				pnp.robotState := 60;
			END_IF;

		60 : (* Wait 200 ms following the ring, then move upward *)
			ton(IN := TRUE);

			IF ton.Q THEN
				tripodGroup.cmd := AxisGroupCmd.MoveLinearRelative;
				tripodGroup.endPoint.c.X := 0;
				tripodGroup.endPoint.c.Y := 0;
				tripodGroup.endPoint.c.Z := 150;
				tripodGroup.coordinateSystem := SM3_Robotics.SMC_COORD_SYSTEM.WCS;
				tripodGroup.bufferMode := SM3_Basic.MC_BUFFER_MODE.Buffered;
				tripodGroup.transitionMode := SM3_Robotics.MC_TRANSITION_MODE.TMNone;
				tripodGroup.transitionParameter := 0;
				pnp.robotState := 70;
			END_IF;

		70 : (* Queue MoveLinearAbsolute to rest (WCS), matching the sample's buffered handoff *)
			tripodGroup.cmd := AxisGroupCmd.MoveLinearAbsolute;
			tripodGroup.endPoint := posRestWCS;
			tripodGroup.coordinateSystem := SM3_Robotics.SMC_COORD_SYSTEM.WCS;
			tripodGroup.bufferMode := SM3_Basic.MC_BUFFER_MODE.BlendingHigh;
			tripodGroup.transitionMode := SM3_Robotics.MC_TRANSITION_MODE.TMCornerDistance;
			tripodGroup.transitionParameter := 500;
			pnp.robotState := 80;

		80 : (* [release] wait rest-pos done; then move above cone (PCS_2) *)
			IF tripodGroup.commandExecuted THEN
				tripodGroup.cmd := AxisGroupCmd.Idle;
			ELSIF tripodGroup.ready THEN
				pnp.targetConePtr := pnp.activeConePtr;
				tripodGroup.cmd := AxisGroupCmd.MoveLinearAbsolute;
				tripodGroup.endPoint := posAboveConePCS2;
				tripodGroup.coordinateSystem := SM3_Robotics.SMC_COORD_SYSTEM.PCS_2;
				tripodGroup.bufferMode := SM3_Basic.MC_BUFFER_MODE.aborting;
				tripodGroup.transitionMode := SM3_Robotics.MC_TRANSITION_MODE.TMNone;
				tripodGroup.transitionParameter := 0;
				pnp.robotState := 90;
			END_IF;

		90 : (* [release] wait above-cone done; then move down to cone (PCS_2) *)
			IF tripodGroup.commandExecuted THEN
				tripodGroup.cmd := AxisGroupCmd.Idle;
			ELSIF tripodGroup.ready THEN
				tripodGroup.cmd := AxisGroupCmd.MoveLinearAbsolute;
				tripodGroup.endPoint := posOnConePCS2;
				tripodGroup.coordinateSystem := SM3_Robotics.SMC_COORD_SYSTEM.PCS_2;
				tripodGroup.bufferMode := SM3_Basic.MC_BUFFER_MODE.aborting;
				tripodGroup.transitionMode := SM3_Robotics.MC_TRANSITION_MODE.TMNone;
				tripodGroup.transitionParameter := 0;
				pnp.robotState := 100;
			END_IF;

		100 : (* [release] ring placed on cone; move back above cone (PCS_2) *)
			IF tripodGroup.commandExecuted THEN
				tripodGroup.cmd := AxisGroupCmd.Idle;
			ELSIF tripodGroup.ready THEN
				tripodGroup.cmd := AxisGroupCmd.MoveLinearAbsolute;
				tripodGroup.endPoint := posAboveConePCS2;
				tripodGroup.coordinateSystem := SM3_Robotics.SMC_COORD_SYSTEM.PCS_2;
				tripodGroup.bufferMode := SM3_Basic.MC_BUFFER_MODE.Buffered;
				tripodGroup.transitionMode := SM3_Robotics.MC_TRANSITION_MODE.TMNone;
				tripodGroup.transitionParameter := 0;
				pnp.robotState := 110;
			END_IF;

		110 : (* [release] wait above-cone done; move back to rest (WCS) *)
			IF tripodGroup.commandExecuted THEN
				tripodGroup.cmd := AxisGroupCmd.Idle;
			ELSIF tripodGroup.ready THEN
				tripodGroup.cmd := AxisGroupCmd.MoveLinearAbsolute;
				tripodGroup.endPoint := posRestWCS;
				tripodGroup.coordinateSystem := SM3_Robotics.SMC_COORD_SYSTEM.WCS;
				tripodGroup.bufferMode := SM3_Basic.MC_BUFFER_MODE.aborting;
				tripodGroup.transitionMode := SM3_Robotics.MC_TRANSITION_MODE.TMNone;
				tripodGroup.transitionParameter := 0;
				pnp.robotState := 120;
			END_IF;

		120 : (* [release] cycle complete; loop to state 40 *)
			IF tripodGroup.commandExecuted THEN
				tripodGroup.cmd := AxisGroupCmd.Idle;
			ELSIF tripodGroup.ready THEN
				pnp.robotState := 40;
			END_IF;
	END_CASE;

	(* Mirror TCP position to shared parameters *)
	pnp.tripodActualPos := tripodGroup.actualPosition;

	(* Status flags (read by Ring and Cone) *)
	pnp.readyForMotion := NOT tripodGroup.groupError AND tripodGroup.status <> AxisGroupStatus.Disabled;
	pnp.ringAttached := pnp.robotState >= 70 AND pnp.robotState <= 100;
	pnp.dontChangePCS_2 := pnp.robotState >= 90 AND pnp.robotState <= 110;

	groupError := tripodGroup.groupError;
	groupErrorId := tripodGroup.groupErrorId;

	(* Auto-reset: rising edge on first scan groupError is TRUE triggers MC_GroupReset -> Standby *)
	tripodGroup.reset := tripodGroup.groupError;

	(* Individual tripod axes *)
	tripodAxis1(
		slave := Tripod1,
		axisEnable := pnp.tripod1Enable,
		cmd := tripodAxis1.cmd,
		position := tripodAxis1.position,
		velocity := tripodVelocity,
		acceleration := tripodAcceleration,
		deceleration := tripodAcceleration,
		jerk := tripodJerk);

	tripodAxis2(
		slave := Tripod2,
		axisEnable := pnp.tripod2Enable,
		cmd := tripodAxis2.cmd,
		position := tripodAxis2.position,
		velocity := tripodVelocity,
		acceleration := tripodAcceleration,
		deceleration := tripodAcceleration,
		jerk := tripodJerk);

	tripodAxis3(
		slave := Tripod3,
		axisEnable := pnp.tripod3Enable,
		cmd := tripodAxis3.cmd,
		position := tripodAxis3.position,
		velocity := tripodVelocity,
		acceleration := tripodAcceleration,
		deceleration := tripodAcceleration,
		jerk := tripodJerk);

	(* Coordinated tripod group - AxisGroup.pou *)
	tripodGroup(
		axisGroupId := 'Tripod',
		axisGroupName := 'Tripod',
		group := Tripod,
		groupEnable := pnp.tripodEnable);

	(* Coordinate transform - called every scan so the FB processes its internal state machine *)
	setCoord(AxisGroup := Tripod);
	END_FUNCTION_BLOCK

(* ---- PickAndPlaceTestSuite.pou ---- *)
(*#-#-#-#-#-#-#-#-#-#---Declaration---#-#-#-#-#-#-#-#-#-#-#-#-#*)

{attribute 'no_assign'}
(*
 * PickAndPlaceTestSuite - integration test suite for a pick-and-place scenario.
 *
 * This test suite directly instantiates and drives the four component controllers:
 *   Environment - drives + cone/ring frame-tracking
 *   TripodRobot - tripod FSM via AxisGroup + Axis wrappers
 *   (Ring and Cone are internal to Environment)
 *
 * Orchestration rules:
 *   operationType = Init -> reset all pnp enable/status flags; no FB calls
 *   operationType = Run -> call TripodRobot then Environment each scan
 *   enable = FALSE -> return immediately, state unchanged
 *
 * Test sequence (20 pass flags):
 *   pass[1] : Init resets all pnp flags; robotState = 0
 *   pass[2] : enable=FALSE leaves robotState unchanged
 *   pass[3] : axis enables set on first Run scan
 *   pass[4] : axes powered/homed; robotState = 10
 *   pass[5] : SetPosition done; robotState = 20
 *   pass[6] : coord transform applied; coordTransformDone; robotState = 30
 *   pass[7] : tripodGroupEnable = TRUE (state 30)
 *   pass[8] : group Standby; robotState = 40
 *   pass[9] : readyForMotion = TRUE at state 40
 *   pass[10] : ringOnTable = TRUE (ring FSM -> state 20)
 *   pass[11] : MoveLinearAbsolute to ring issued; robotState = 50
 *   pass[12] : arrived at ring; robotState = 60
 *   pass[13] : up from ring (200 ms TON); robotState = 70
 *   pass[14] : ringAttached = TRUE (robotState in [70..100])
 *   pass[15] : rest position; robotState = 80
 *   pass[16] : above cone; robotState = 90
 *   pass[17] : dontChangePCS_2 = TRUE (robotState in [90..110])
 *   pass[18] : ring on cone; robotState = 100
 *   pass[19] : up from cone; robotState = 110
 *   pass[20] : cycle complete; robotState loops back to 40
 *)
PROGRAM PickAndPlaceTestSuite
VAR_EXTERNAL
	pnp : PickAndPlaceFixture;
END_VAR
VAR CONSTANT
	TIMEOUT : UDINT  := 5000;
END_VAR
VAR
	(* Component controllers *)
	env : Environment;
	tripodRobot : TripodRobot;

	(* Orchestration control - set by test steps each scan *)
	operationType : OperatingMode := OperatingMode.Init;
	enable : BOOL;

	(* Orchestration outputs *)
	error : BOOL;
	done : BOOL;

	(* Test infrastructure *)
	step : UINT  := 0;
	cycles : UDINT := 0;
	testDone : BOOL;
	testFailed : BOOL;
	failStep : UINT;
	testReset : BOOL;
	allPass : BOOL;
	pass : ARRAY[1..20] OF BOOL;

	(* Diagnostic mirrors - inspect when testFailed = TRUE *)
	mirRobotState : INT;
	mirAxis1Enable : BOOL;
	mirAxis2Enable : BOOL;
	mirAxis3Enable : BOOL;
	mirGroupEnable : BOOL;
	mirCoordTransformOk : BOOL;
	mirReadyForMotion : BOOL;
	mirRingAttached : BOOL;
	mirDontChangePCS2 : BOOL;
	mirRingOnTable : BOOL;
	mirError : BOOL;
	i : UINT;
END_VAR

(*#-#-#-#-#-#-#-#-#-#---Implementation---#-#-#-#-#-#-#-#-#-#-#-#-#*)

(* Watchdog - timeout *)
cycles := cycles + 1;
IF (cycles > TIMEOUT) AND NOT testDone THEN
	testFailed := TRUE;
	failStep   := step;
END_IF;

(* Watchdog - group error *)
IF error AND NOT testDone THEN
	testFailed := TRUE;
	failStep   := step;
END_IF;

(* Post-failure cleanup - run Init every scan to power down drives cleanly *)
IF testFailed THEN
	PickAndPlaceData.pnp.tripod1Enable := FALSE;
	PickAndPlaceData.pnp.tripod2Enable := FALSE;
	PickAndPlaceData.pnp.tripod3Enable := FALSE;
	PickAndPlaceData.pnp.tripodEnable := FALSE;
	PickAndPlaceData.pnp.rotaryTableEnable := FALSE;
	PickAndPlaceData.pnp.conveyorEnable := FALSE;
	PickAndPlaceData.pnp.coordTransformDone := FALSE;
	PickAndPlaceData.pnp.robotState := 0;
	PickAndPlaceData.pnp.readyForMotion := FALSE;
	PickAndPlaceData.pnp.ringAttached := FALSE;
	PickAndPlaceData.pnp.dontChangePCS_2 := FALSE;
	PickAndPlaceData.pnp.ringOnTable := FALSE;
	env(operationType := OperatingMode.Init);
	tripodRobot(operationType := OperatingMode.Init);
	RETURN;
END_IF;

(* Warm-download reset - write testReset := TRUE in the online monitor *)
IF testReset THEN
	step := 0;
	cycles := 0;
	testDone := FALSE;
	testFailed := FALSE;
	failStep := 0;
	allPass := FALSE;
	FOR i := 1 TO 20 DO pass[i] := FALSE; END_FOR;
	testReset := FALSE;
END_IF;

(*
 * Test sequence
 *
 * Each step sets operationType / enable for this scan, then checks the
 * result of the previous scan's orchestration (at the bottom of this POU body).
 * Motion steps take many cycles; the TIMEOUT watchdog is the safety net.
 * cycles > 1 guards on steps 4-8 give the drives at
 * least one full orchestration cycle before the state check fires.
 *)
CASE step OF
	0 : (* boot: run Init once to reach a clean known state *)
		operationType := OperatingMode.Init; PickAndPlaceTestSuite.enable := TRUE;
		step := 1; cycles := 0;

	(* pass[1] - Init resets all pap flags *)
	1 :
		operationType := OperatingMode.Init; PickAndPlaceTestSuite.enable := TRUE;
		IF NOT PickAndPlaceData.pnp.tripod1Enable
				AND NOT PickAndPlaceData.pnp.tripod2Enable
				AND NOT PickAndPlaceData.pnp.tripod3Enable
		   		AND NOT PickAndPlaceData.pnp.tripodEnable
		   		AND NOT PickAndPlaceData.pnp.rotaryTableEnable
		   		AND NOT PickAndPlaceData.pnp.conveyorEnable
		   		AND NOT PickAndPlaceData.pnp.coordTransformDone
		   		AND (PickAndPlaceData.pnp.robotState = 0)
		   		AND NOT PickAndPlaceData.pnp.readyForMotion
		   		AND NOT PickAndPlaceData.pnp.ringAttached
		   		AND NOT PickAndPlaceData.pnp.dontChangePCS_2
		   		AND NOT PickAndPlaceData.pnp.ringOnTable THEN
			pass[1] := TRUE;
			step := 2; cycles := 0;
		END_IF;

	(* pass[2] - enable=FALSE leaves robotState unchanged *)
	2 :
		operationType := OperatingMode.Run; PickAndPlaceTestSuite.enable := FALSE;
		IF cycles > 1 AND PickAndPlaceData.pnp.robotState = 0 THEN
			pass[2] := TRUE;
			operationType := OperatingMode.Init; PickAndPlaceTestSuite.enable := TRUE;
			PickAndPlaceData.pnp.automaticPnp := TRUE;
			step := 3; cycles := 0;
		END_IF;

	(* pass[3] - axis enable flags set on the first Run scan *)
	3 :
		operationType := OperatingMode.Run; PickAndPlaceTestSuite.enable := TRUE;
		IF cycles > 0 AND PickAndPlaceData.pnp.tripod1Enable
				AND PickAndPlaceData.pnp.tripod2Enable
				AND PickAndPlaceData.pnp.tripod3Enable THEN
			pass[3] := TRUE;
			step := 4; cycles := 0;
		END_IF;

	(* pass[4] - all three tripod axes powered and homed; robotState = 10 *)
	4 :
		operationType := OperatingMode.Run; PickAndPlaceTestSuite.enable := TRUE;
		IF cycles > 1 AND PickAndPlaceData.pnp.robotState = 10 THEN
			pass[4] := TRUE;
			step := 5; cycles := 0;
		END_IF;

	(* pass[5] - SetPosition done for all three axes; robotState = 20 *)
	5 :
		operationType := OperatingMode.Run; PickAndPlaceTestSuite.enable := TRUE;
		IF cycles > 1 AND PickAndPlaceData.pnp.robotState = 20 THEN
			pass[5] := TRUE;
			step := 6; cycles := 0;
		END_IF;

	(* pass[6] - coordinate transform applied; bCoordTransformOk = TRUE; robotState = 30 *)
	6 :
		operationType := OperatingMode.Run; PickAndPlaceTestSuite.enable := TRUE;
		IF cycles > 1 AND PickAndPlaceData.pnp.coordTransformDone
				AND PickAndPlaceData.pnp.robotState = 30 THEN
			pass[6] := TRUE;
			step := 7; cycles := 0;
		END_IF;

	(* pass[7] - tripodGroupEnable = TRUE *)
	7 :
		operationType := OperatingMode.Run; PickAndPlaceTestSuite.enable := TRUE;
		IF cycles > 1 AND PickAndPlaceData.pnp.tripodEnable THEN
			pass[7] := TRUE;
			step := 8; cycles := 0;
		END_IF;

	(* pass[8] - axis group in Standby; robotState = 40 *)
	8 :
		operationType := OperatingMode.Run; PickAndPlaceTestSuite.enable := TRUE;
		IF cycles > 1 AND PickAndPlaceData.pnp.robotState = 40 THEN
			pass[8] := TRUE;
			step := 9; cycles := 0;
		END_IF;

	(* pass[9] - bReadyForMotion = TRUE at state 40 *)
	9 :
		operationType := OperatingMode.Run; PickAndPlaceTestSuite.enable := TRUE;
		IF PickAndPlaceData.pnp.readyForMotion THEN
			pass[9] := TRUE;
			step := 10; cycles := 0;
		END_IF

	(* pass[10] - bRingOnTable = TRUE (ring FSM -> state 20) *)
	10 :
		operationType := OperatingMode.Run; PickAndPlaceTestSuite.enable := TRUE;
		IF PickAndPlaceData.pnp.ringOnTable THEN
			pass[10] := TRUE;
			step := 11; cycles := 0;
		END_IF;

	(* pass[11] - MoveLinearAbsolute to ring issued; robotState = 50 *)
	11 :
		operationType := OperatingMode.Run; PickAndPlaceTestSuite.enable := TRUE;
		IF PickAndPlaceData.pnp.robotState = 50 THEN
			pass[11] := TRUE;
			step := 12; cycles := 0;
		END_IF;

	(* pass[12] - arrived at ring; robotState = 60 *)
	12 :
		operationType := OperatingMode.Run; PickAndPlaceTestSuite.enable := TRUE;
		IF PickAndPlaceData.pnp.robotState = 60 THEN
			pass[12] := TRUE;
			step := 13; cycles := 0;
		END_IF;

	(* pass[13] - up from ring (200 ms TON elapsed); robotState = 70 *)
	13 :
		operationType := OperatingMode.Run; PickAndPlaceTestSuite.enable := TRUE;
		IF PickAndPlaceData.pnp.robotState = 70 THEN
			pass[13] := TRUE;
			step := 14; cycles := 0;
		END_IF;

	(* pass[14] - bRingAttached = TRUE while robotState in [70..100] *)
	14 :
		operationType := OperatingMode.Run; PickAndPlaceTestSuite.enable := TRUE;
		IF PickAndPlaceData.pnp.ringAttached AND PickAndPlaceData.pnp.robotState >= 70
				AND PickAndPlaceData.pnp.robotState <= 100 THEN
			pass[14] := TRUE;
			step := 15; cycles := 0;
		END_IF;

	(* pass[15] - robot at WCS rest position; robotState = 80 *)
	15 :
		operationType := OperatingMode.Run; PickAndPlaceTestSuite.enable := TRUE;
		IF PickAndPlaceData.pnp.robotState = 80 THEN
			pass[15] := TRUE;
			step := 16; cycles := 0;
		END_IF;

	(* pass[16] - robot above cone (PCS_2); robotState = 90 *)
	16 :
		operationType := OperatingMode.Run; PickAndPlaceTestSuite.enable := TRUE;
		IF PickAndPlaceData.pnp.robotState = 90 THEN
			pass[16] := TRUE;
			step := 17; cycles := 0;
		END_IF;

	(* pass[17] - bDontChangePCS_2 = TRUE while robotState in [90..110] *)
	17 :
		operationType := OperatingMode.Run; PickAndPlaceTestSuite.enable := TRUE;
		IF PickAndPlaceData.pnp.dontChangePCS_2 AND PickAndPlaceData.pnp.robotState >= 90
				AND PickAndPlaceData.pnp.robotState <= 110 THEN
			pass[17] := TRUE;
			step := 18; cycles := 0;
		END_IF;

	(* pass[18] - ring placed on cone; robotState = 100 *)
	18 :
		operationType := OperatingMode.Run; PickAndPlaceTestSuite.enable := TRUE;
		IF PickAndPlaceData.pnp.robotState = 100 THEN
			pass[18] := TRUE;
			step := 19; cycles := 0;
		END_IF;

	(* pass[19] - up from cone; robotState = 110; bDontChangePCS_2 still TRUE *)
	19 :
		operationType := OperatingMode.Run; PickAndPlaceTestSuite.enable := TRUE;
		IF PickAndPlaceData.pnp.robotState = 110 AND PickAndPlaceData.pnp.dontChangePCS_2 THEN
			pass[19] := TRUE;
			step := 20; cycles := 0;
		END_IF;

	(* pass[20] - cycle complete; robotState loops back to 40 *)
	20 :
		operationType := OperatingMode.Run; PickAndPlaceTestSuite.enable := TRUE;
		IF PickAndPlaceData.pnp.robotState = 40 AND pass[18] AND pass[19] THEN
			pass[20] := TRUE;
			testDone := TRUE;
			step := 21; cycles := 0;
		END_IF;
END_CASE;

(* Summary flag *)
allPass := pass[1] AND pass[2] AND pass[3] AND pass[4] AND pass[5]
	AND pass[6] AND pass[7] AND pass[8] AND pass[9] AND pass[10]
    AND pass[11] AND pass[12] AND pass[13] AND pass[14] AND pass[15]
    AND pass[16] AND pass[17] AND pass[18] AND pass[19] AND pass[20];

(* Diagnostic mirrors *)
mirRobotState := PickAndPlaceData.pnp.robotState;
mirAxis1Enable := PickAndPlaceData.pnp.tripod1Enable;
mirAxis2Enable := PickAndPlaceData.pnp.tripod2Enable;
mirAxis3Enable := PickAndPlaceData.pnp.tripod3Enable;
mirGroupEnable := PickAndPlaceData.pnp.tripodEnable;
mirCoordTransformOk := PickAndPlaceData.pnp.coordTransformDone;
mirReadyForMotion := PickAndPlaceData.pnp.readyForMotion;
mirRingAttached := PickAndPlaceData.pnp.ringAttached;
mirDontChangePCS2 := PickAndPlaceData.pnp.dontChangePCS_2;
mirRingOnTable := PickAndPlaceData.pnp.ringOnTable;
mirError := error;

IF NOT PickAndPlaceTestSuite.enable THEN
	(* nothing - state frozen *)
ELSIF operationType = OperatingMode.Init THEN
	PickAndPlaceData.pnp.tripod1Enable := FALSE;
	PickAndPlaceData.pnp.tripod2Enable := FALSE;
	PickAndPlaceData.pnp.tripod3Enable := FALSE;
	PickAndPlaceData.pnp.tripodEnable := FALSE;
	PickAndPlaceData.pnp.rotaryTableEnable := FALSE;
	PickAndPlaceData.pnp.conveyorEnable := FALSE;
	PickAndPlaceData.pnp.coordTransformDone := FALSE;
	PickAndPlaceData.pnp.robotState := 0;
	PickAndPlaceData.pnp.readyForMotion := FALSE;
	PickAndPlaceData.pnp.ringAttached := FALSE;
	PickAndPlaceData.pnp.dontChangePCS_2 := FALSE;
	PickAndPlaceData.pnp.ringOnTable := FALSE;
ELSE
	tripodRobot(operationType := operationType);
	env(operationType := operationType);
END_IF;

error := tripodRobot.groupError;
done := PickAndPlaceData.pnp.robotState >= 120 AND NOT tripodRobot.groupError;

(* ---- PickAndPlaceTestSuite.st ---- *)
(*
 * PickAndPlaceTestSuite - integration test suite for a pick-and-place scenario.
 *
 * This test suite directly instantiates and drives the four component controllers:
 *   Environment - drives + cone/ring frame-tracking
 *   TripodRobot - tripod FSM via AxisGroup + Axis wrappers
 *   (Ring and Cone are internal to Environment)
 *
 * Orchestration rules:
 *   operationType = Init -> reset all pnp enable/status flags; no FB calls
 *   operationType = Run -> call TripodRobot then Environment each scan
 *   enable = FALSE -> return immediately, state unchanged
 *
 * Test sequence (20 pass flags):
 *   pass[1] : Init resets all pnp flags; robotState = 0
 *   pass[2] : enable=FALSE leaves robotState unchanged
 *   pass[3] : axis enables set on first Run scan
 *   pass[4] : axes powered/homed; robotState = 10
 *   pass[5] : SetPosition done; robotState = 20
 *   pass[6] : coord transform applied; coordTransformDone; robotState = 30
 *   pass[7] : tripodGroupEnable = TRUE (state 30)
 *   pass[8] : group Standby; robotState = 40
 *   pass[9] : readyForMotion = TRUE at state 40
 *   pass[10] : ringOnTable = TRUE (ring FSM -> state 20)
 *   pass[11] : MoveLinearAbsolute to ring issued; robotState = 50
 *   pass[12] : arrived at ring; robotState = 60
 *   pass[13] : up from ring (200 ms TON); robotState = 70
 *   pass[14] : ringAttached = TRUE (robotState in [70..100])
 *   pass[15] : rest position; robotState = 80
 *   pass[16] : above cone; robotState = 90
 *   pass[17] : dontChangePCS_2 = TRUE (robotState in [90..110])
 *   pass[18] : ring on cone; robotState = 100
 *   pass[19] : up from cone; robotState = 110
 *   pass[20] : cycle complete; robotState loops back to 40
 *)
PROGRAM PickAndPlaceTestSuite
	VAR_EXTERNAL
		pnp : PickAndPlaceFixture;
	END_VAR
	VAR CONSTANT
		TIMEOUT : UDINT  := 5000;
	END_VAR
	VAR
		(* Component controllers *)
		env : Environment;
		tripodRobot : TripodRobot;

		(* Orchestration control - set by test steps each scan *)
		operationType : OperatingMode := OperatingMode.Init;
		enable : BOOL;

		(* Orchestration outputs *)
		error : BOOL;
		done : BOOL;

		(* Test infrastructure *)
		step : UINT  := 0;
		cycles : UDINT := 0;
		testDone : BOOL;
		testFailed : BOOL;
		failStep : UINT;
		testReset : BOOL;
		allPass : BOOL;
		pass : ARRAY[1..20] OF BOOL;

		(* Diagnostic mirrors - inspect when testFailed = TRUE *)
		mirRobotState : INT;
		mirAxis1Enable : BOOL;
		mirAxis2Enable : BOOL;
		mirAxis3Enable : BOOL;
		mirGroupEnable : BOOL;
		mirCoordTransformOk : BOOL;
		mirReadyForMotion : BOOL;
		mirRingAttached : BOOL;
		mirDontChangePCS2 : BOOL;
		mirRingOnTable : BOOL;
		mirError : BOOL;
		i : UINT;
	END_VAR

	(* Watchdog - timeout *)
	cycles := cycles + 1;
	IF (cycles > TIMEOUT) AND NOT testDone THEN
		testFailed := TRUE;
		failStep   := step;
	END_IF;

	(* Watchdog - group error *)
	IF error AND NOT testDone THEN
		testFailed := TRUE;
		failStep   := step;
	END_IF;

	(* Post-failure cleanup - run Init every scan to power down drives cleanly *)
	IF testFailed THEN
		PickAndPlaceData.pnp.tripod1Enable := FALSE;
		PickAndPlaceData.pnp.tripod2Enable := FALSE;
		PickAndPlaceData.pnp.tripod3Enable := FALSE;
		PickAndPlaceData.pnp.tripodEnable := FALSE;
		PickAndPlaceData.pnp.rotaryTableEnable := FALSE;
		PickAndPlaceData.pnp.conveyorEnable := FALSE;
		PickAndPlaceData.pnp.coordTransformDone := FALSE;
		PickAndPlaceData.pnp.robotState := 0;
		PickAndPlaceData.pnp.readyForMotion := FALSE;
		PickAndPlaceData.pnp.ringAttached := FALSE;
		PickAndPlaceData.pnp.dontChangePCS_2 := FALSE;
		PickAndPlaceData.pnp.ringOnTable := FALSE;
		env(operationType := OperatingMode.Init);
		tripodRobot(operationType := OperatingMode.Init);
		RETURN;
	END_IF;

	(* Warm-download reset - write testReset := TRUE in the online monitor *)
	IF testReset THEN
		step := 0;
		cycles := 0;
		testDone := FALSE;
		testFailed := FALSE;
		failStep := 0;
		allPass := FALSE;
		FOR i := 1 TO 20 DO pass[i] := FALSE; END_FOR;
		testReset := FALSE;
	END_IF;

	(*
	 * Test sequence
	 *
	 * Each step sets operationType / enable for this scan, then checks the
	 * result of the previous scan's orchestration (at the bottom of this POU body).
	 * Motion steps take many cycles; the TIMEOUT watchdog is the safety net.
	 * cycles > 1 guards on steps 4-8 give the drives at
	 * least one full orchestration cycle before the state check fires.
	 *)
	CASE step OF
		0 : (* boot: run Init once to reach a clean known state *)
			operationType := OperatingMode.Init; PickAndPlaceTestSuite.enable := TRUE;
			step := 1; cycles := 0;

		(* pass[1] - Init resets all pap flags *)
		1 :
			operationType := OperatingMode.Init; PickAndPlaceTestSuite.enable := TRUE;
			IF NOT PickAndPlaceData.pnp.tripod1Enable
					AND NOT PickAndPlaceData.pnp.tripod2Enable
					AND NOT PickAndPlaceData.pnp.tripod3Enable
			   		AND NOT PickAndPlaceData.pnp.tripodEnable
			   		AND NOT PickAndPlaceData.pnp.rotaryTableEnable
			   		AND NOT PickAndPlaceData.pnp.conveyorEnable
			   		AND NOT PickAndPlaceData.pnp.coordTransformDone
			   		AND (PickAndPlaceData.pnp.robotState = 0)
			   		AND NOT PickAndPlaceData.pnp.readyForMotion
			   		AND NOT PickAndPlaceData.pnp.ringAttached
			   		AND NOT PickAndPlaceData.pnp.dontChangePCS_2
			   		AND NOT PickAndPlaceData.pnp.ringOnTable THEN
				pass[1] := TRUE;
				step := 2; cycles := 0;
			END_IF;

		(* pass[2] - enable=FALSE leaves robotState unchanged *)
		2 :
			operationType := OperatingMode.Run; PickAndPlaceTestSuite.enable := FALSE;
			IF cycles > 1 AND PickAndPlaceData.pnp.robotState = 0 THEN
				pass[2] := TRUE;
				operationType := OperatingMode.Init; PickAndPlaceTestSuite.enable := TRUE;
				PickAndPlaceData.pnp.automaticPnp := TRUE;
				step := 3; cycles := 0;
			END_IF;

		(* pass[3] - axis enable flags set on the first Run scan *)
		3 :
			operationType := OperatingMode.Run; PickAndPlaceTestSuite.enable := TRUE;
			IF cycles > 0 AND PickAndPlaceData.pnp.tripod1Enable
					AND PickAndPlaceData.pnp.tripod2Enable
					AND PickAndPlaceData.pnp.tripod3Enable THEN
				pass[3] := TRUE;
				step := 4; cycles := 0;
			END_IF;

		(* pass[4] - all three tripod axes powered and homed; robotState = 10 *)
		4 :
			operationType := OperatingMode.Run; PickAndPlaceTestSuite.enable := TRUE;
			IF cycles > 1 AND PickAndPlaceData.pnp.robotState = 10 THEN
				pass[4] := TRUE;
				step := 5; cycles := 0;
			END_IF;

		(* pass[5] - SetPosition done for all three axes; robotState = 20 *)
		5 :
			operationType := OperatingMode.Run; PickAndPlaceTestSuite.enable := TRUE;
			IF cycles > 1 AND PickAndPlaceData.pnp.robotState = 20 THEN
				pass[5] := TRUE;
				step := 6; cycles := 0;
			END_IF;

		(* pass[6] - coordinate transform applied; bCoordTransformOk = TRUE; robotState = 30 *)
		6 :
			operationType := OperatingMode.Run; PickAndPlaceTestSuite.enable := TRUE;
			IF cycles > 1 AND PickAndPlaceData.pnp.coordTransformDone
					AND PickAndPlaceData.pnp.robotState = 30 THEN
				pass[6] := TRUE;
				step := 7; cycles := 0;
			END_IF;

		(* pass[7] - tripodGroupEnable = TRUE *)
		7 :
			operationType := OperatingMode.Run; PickAndPlaceTestSuite.enable := TRUE;
			IF cycles > 1 AND PickAndPlaceData.pnp.tripodEnable THEN
				pass[7] := TRUE;
				step := 8; cycles := 0;
			END_IF;

		(* pass[8] - axis group in Standby; robotState = 40 *)
		8 :
			operationType := OperatingMode.Run; PickAndPlaceTestSuite.enable := TRUE;
			IF cycles > 1 AND PickAndPlaceData.pnp.robotState = 40 THEN
				pass[8] := TRUE;
				step := 9; cycles := 0;
			END_IF;

		(* pass[9] - bReadyForMotion = TRUE at state 40 *)
		9 :
			operationType := OperatingMode.Run; PickAndPlaceTestSuite.enable := TRUE;
			IF PickAndPlaceData.pnp.readyForMotion THEN
				pass[9] := TRUE;
				step := 10; cycles := 0;
			END_IF

		(* pass[10] - bRingOnTable = TRUE (ring FSM -> state 20) *)
		10 :
			operationType := OperatingMode.Run; PickAndPlaceTestSuite.enable := TRUE;
			IF PickAndPlaceData.pnp.ringOnTable THEN
				pass[10] := TRUE;
				step := 11; cycles := 0;
			END_IF;

		(* pass[11] - MoveLinearAbsolute to ring issued; robotState = 50 *)
		11 :
			operationType := OperatingMode.Run; PickAndPlaceTestSuite.enable := TRUE;
			IF PickAndPlaceData.pnp.robotState = 50 THEN
				pass[11] := TRUE;
				step := 12; cycles := 0;
			END_IF;

		(* pass[12] - arrived at ring; robotState = 60 *)
		12 :
			operationType := OperatingMode.Run; PickAndPlaceTestSuite.enable := TRUE;
			IF PickAndPlaceData.pnp.robotState = 60 THEN
				pass[12] := TRUE;
				step := 13; cycles := 0;
			END_IF;

		(* pass[13] - up from ring (200 ms TON elapsed); robotState = 70 *)
		13 :
			operationType := OperatingMode.Run; PickAndPlaceTestSuite.enable := TRUE;
			IF PickAndPlaceData.pnp.robotState = 70 THEN
				pass[13] := TRUE;
				step := 14; cycles := 0;
			END_IF;

		(* pass[14] - bRingAttached = TRUE while robotState in [70..100] *)
		14 :
			operationType := OperatingMode.Run; PickAndPlaceTestSuite.enable := TRUE;
			IF PickAndPlaceData.pnp.ringAttached AND PickAndPlaceData.pnp.robotState >= 70
					AND PickAndPlaceData.pnp.robotState <= 100 THEN
				pass[14] := TRUE;
				step := 15; cycles := 0;
			END_IF;

		(* pass[15] - robot at WCS rest position; robotState = 80 *)
		15 :
			operationType := OperatingMode.Run; PickAndPlaceTestSuite.enable := TRUE;
			IF PickAndPlaceData.pnp.robotState = 80 THEN
				pass[15] := TRUE;
				step := 16; cycles := 0;
			END_IF;

		(* pass[16] - robot above cone (PCS_2); robotState = 90 *)
		16 :
			operationType := OperatingMode.Run; PickAndPlaceTestSuite.enable := TRUE;
			IF PickAndPlaceData.pnp.robotState = 90 THEN
				pass[16] := TRUE;
				step := 17; cycles := 0;
			END_IF;

		(* pass[17] - bDontChangePCS_2 = TRUE while robotState in [90..110] *)
		17 :
			operationType := OperatingMode.Run; PickAndPlaceTestSuite.enable := TRUE;
			IF PickAndPlaceData.pnp.dontChangePCS_2 AND PickAndPlaceData.pnp.robotState >= 90
					AND PickAndPlaceData.pnp.robotState <= 110 THEN
				pass[17] := TRUE;
				step := 18; cycles := 0;
			END_IF;

		(* pass[18] - ring placed on cone; robotState = 100 *)
		18 :
			operationType := OperatingMode.Run; PickAndPlaceTestSuite.enable := TRUE;
			IF PickAndPlaceData.pnp.robotState = 100 THEN
				pass[18] := TRUE;
				step := 19; cycles := 0;
			END_IF;

		(* pass[19] - up from cone; robotState = 110; bDontChangePCS_2 still TRUE *)
		19 :
			operationType := OperatingMode.Run; PickAndPlaceTestSuite.enable := TRUE;
			IF PickAndPlaceData.pnp.robotState = 110 AND PickAndPlaceData.pnp.dontChangePCS_2 THEN
				pass[19] := TRUE;
				step := 20; cycles := 0;
			END_IF;

		(* pass[20] - cycle complete; robotState loops back to 40 *)
		20 :
			operationType := OperatingMode.Run; PickAndPlaceTestSuite.enable := TRUE;
			IF PickAndPlaceData.pnp.robotState = 40 AND pass[18] AND pass[19] THEN
				pass[20] := TRUE;
				testDone := TRUE;
				step := 21; cycles := 0;
			END_IF;
	END_CASE;

	(* Summary flag *)
	allPass := pass[1] AND pass[2] AND pass[3] AND pass[4] AND pass[5]
		AND pass[6] AND pass[7] AND pass[8] AND pass[9] AND pass[10]
	    AND pass[11] AND pass[12] AND pass[13] AND pass[14] AND pass[15]
	    AND pass[16] AND pass[17] AND pass[18] AND pass[19] AND pass[20];

	(* Diagnostic mirrors *)
	mirRobotState := PickAndPlaceData.pnp.robotState;
	mirAxis1Enable := PickAndPlaceData.pnp.tripod1Enable;
	mirAxis2Enable := PickAndPlaceData.pnp.tripod2Enable;
	mirAxis3Enable := PickAndPlaceData.pnp.tripod3Enable;
	mirGroupEnable := PickAndPlaceData.pnp.tripodEnable;
	mirCoordTransformOk := PickAndPlaceData.pnp.coordTransformDone;
	mirReadyForMotion := PickAndPlaceData.pnp.readyForMotion;
	mirRingAttached := PickAndPlaceData.pnp.ringAttached;
	mirDontChangePCS2 := PickAndPlaceData.pnp.dontChangePCS_2;
	mirRingOnTable := PickAndPlaceData.pnp.ringOnTable;
	mirError := error;

	IF NOT PickAndPlaceTestSuite.enable THEN
		(* nothing - state frozen *)
	ELSIF operationType = OperatingMode.Init THEN
		PickAndPlaceData.pnp.tripod1Enable := FALSE;
		PickAndPlaceData.pnp.tripod2Enable := FALSE;
		PickAndPlaceData.pnp.tripod3Enable := FALSE;
		PickAndPlaceData.pnp.tripodEnable := FALSE;
		PickAndPlaceData.pnp.rotaryTableEnable := FALSE;
		PickAndPlaceData.pnp.conveyorEnable := FALSE;
		PickAndPlaceData.pnp.coordTransformDone := FALSE;
		PickAndPlaceData.pnp.robotState := 0;
		PickAndPlaceData.pnp.readyForMotion := FALSE;
		PickAndPlaceData.pnp.ringAttached := FALSE;
		PickAndPlaceData.pnp.dontChangePCS_2 := FALSE;
		PickAndPlaceData.pnp.ringOnTable := FALSE;
	ELSE
		tripodRobot(operationType := operationType);
		env(operationType := operationType);
	END_IF;

	error := tripodRobot.groupError;
	done := PickAndPlaceData.pnp.robotState >= 120 AND NOT tripodRobot.groupError;
	END_PROGRAM

(* ---- TestTripodPlanning.st ---- *)
PROGRAM TestTripodPlanning

	;
	END_PROGRAM
